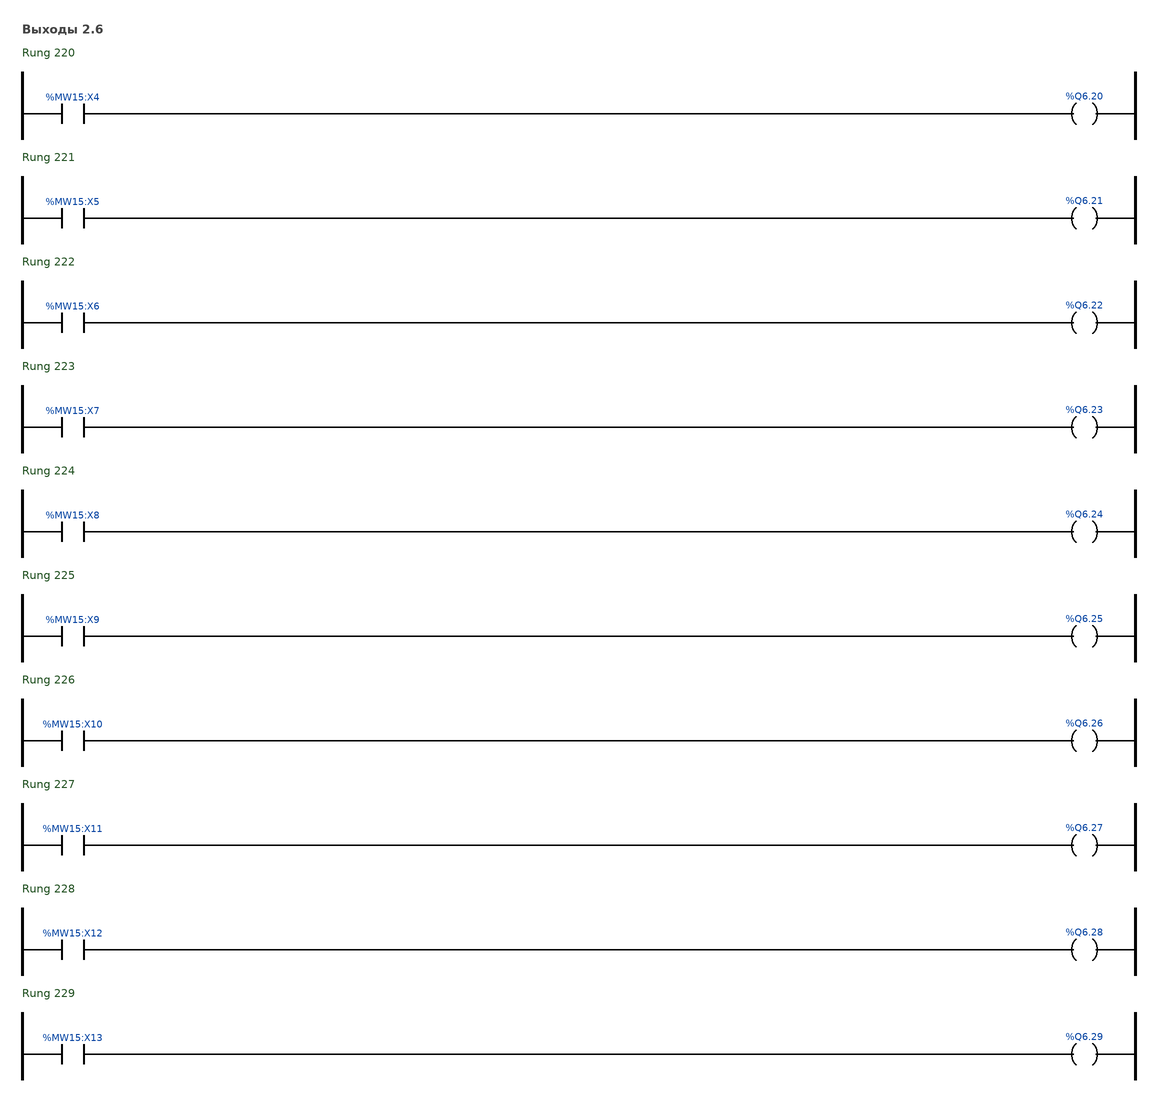

// Rung 220
  LD %MW15:X4
  ST %Q6.20
  // as ST:
  //   %Q6.20 := %MW15:X4;

// Rung 221
  LD %MW15:X5
  ST %Q6.21
  // as ST:
  //   %Q6.21 := %MW15:X5;

// Rung 222
  LD %MW15:X6
  ST %Q6.22
  // as ST:
  //   %Q6.22 := %MW15:X6;

// Rung 223
  LD %MW15:X7
  ST %Q6.23
  // as ST:
  //   %Q6.23 := %MW15:X7;

// Rung 224
  LD %MW15:X8
  ST %Q6.24
  // as ST:
  //   %Q6.24 := %MW15:X8;

// Rung 225
  LD %MW15:X9
  ST %Q6.25
  // as ST:
  //   %Q6.25 := %MW15:X9;

// Rung 226
  LD %MW15:X10
  ST %Q6.26
  // as ST:
  //   %Q6.26 := %MW15:X10;

// Rung 227
  LD %MW15:X11
  ST %Q6.27
  // as ST:
  //   %Q6.27 := %MW15:X11;

// Rung 228
  LD %MW15:X12
  ST %Q6.28
  // as ST:
  //   %Q6.28 := %MW15:X12;

// Rung 229
  LD %MW15:X13
  ST %Q6.29
  // as ST:
  //   %Q6.29 := %MW15:X13;

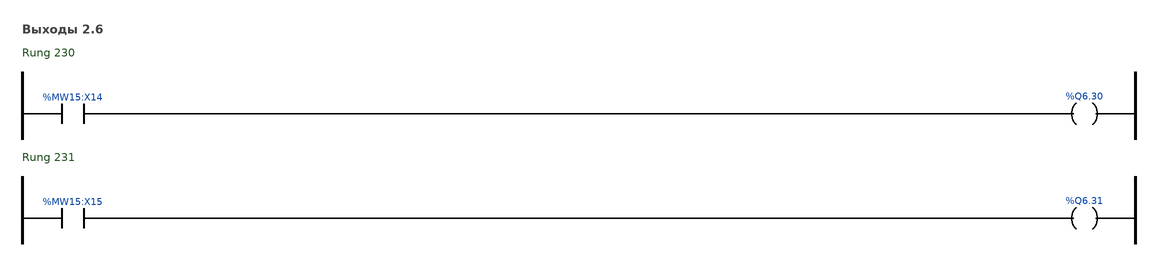

// Rung 230
  LD %MW15:X14
  ST %Q6.30
  // as ST:
  //   %Q6.30 := %MW15:X14;

// Rung 231
  LD %MW15:X15
  ST %Q6.31
  // as ST:
  //   %Q6.31 := %MW15:X15;

POU Выходы 2.7
  (* SectionNumber=9 *)

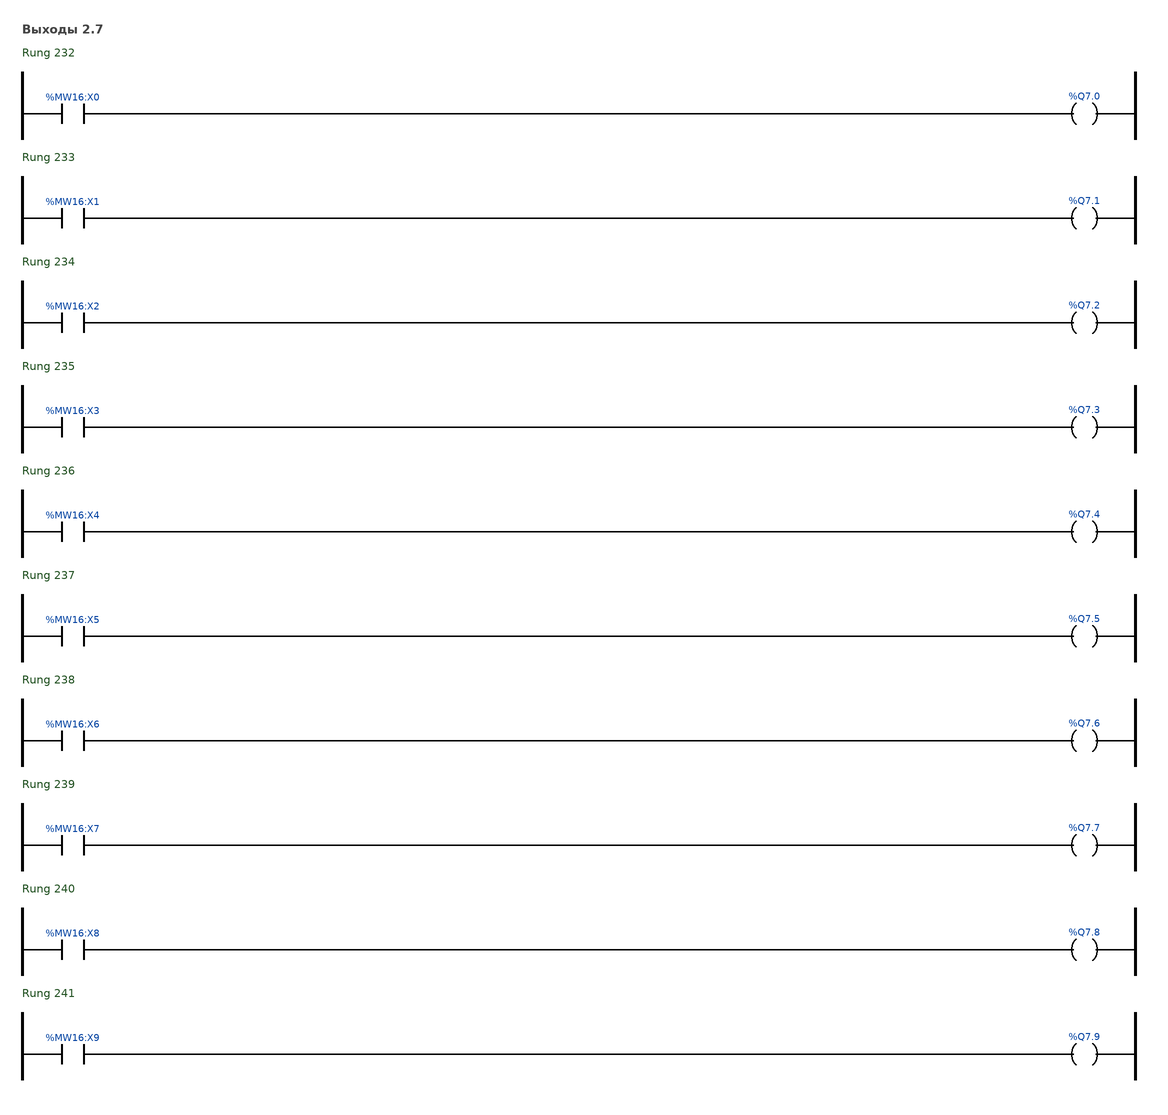

// Rung 232
  LD %MW16:X0
  ST %Q7.0
  // as ST:
  //   %Q7.0 := %MW16:X0;

// Rung 233
  LD %MW16:X1
  ST %Q7.1
  // as ST:
  //   %Q7.1 := %MW16:X1;

// Rung 234
  LD %MW16:X2
  ST %Q7.2
  // as ST:
  //   %Q7.2 := %MW16:X2;

// Rung 235
  LD %MW16:X3
  ST %Q7.3
  // as ST:
  //   %Q7.3 := %MW16:X3;

// Rung 236
  LD %MW16:X4
  ST %Q7.4
  // as ST:
  //   %Q7.4 := %MW16:X4;

// Rung 237
  LD %MW16:X5
  ST %Q7.5
  // as ST:
  //   %Q7.5 := %MW16:X5;

// Rung 238
  LD %MW16:X6
  ST %Q7.6
  // as ST:
  //   %Q7.6 := %MW16:X6;

// Rung 239
  LD %MW16:X7
  ST %Q7.7
  // as ST:
  //   %Q7.7 := %MW16:X7;

// Rung 240
  LD %MW16:X8
  ST %Q7.8
  // as ST:
  //   %Q7.8 := %MW16:X8;

// Rung 241
  LD %MW16:X9
  ST %Q7.9
  // as ST:
  //   %Q7.9 := %MW16:X9;

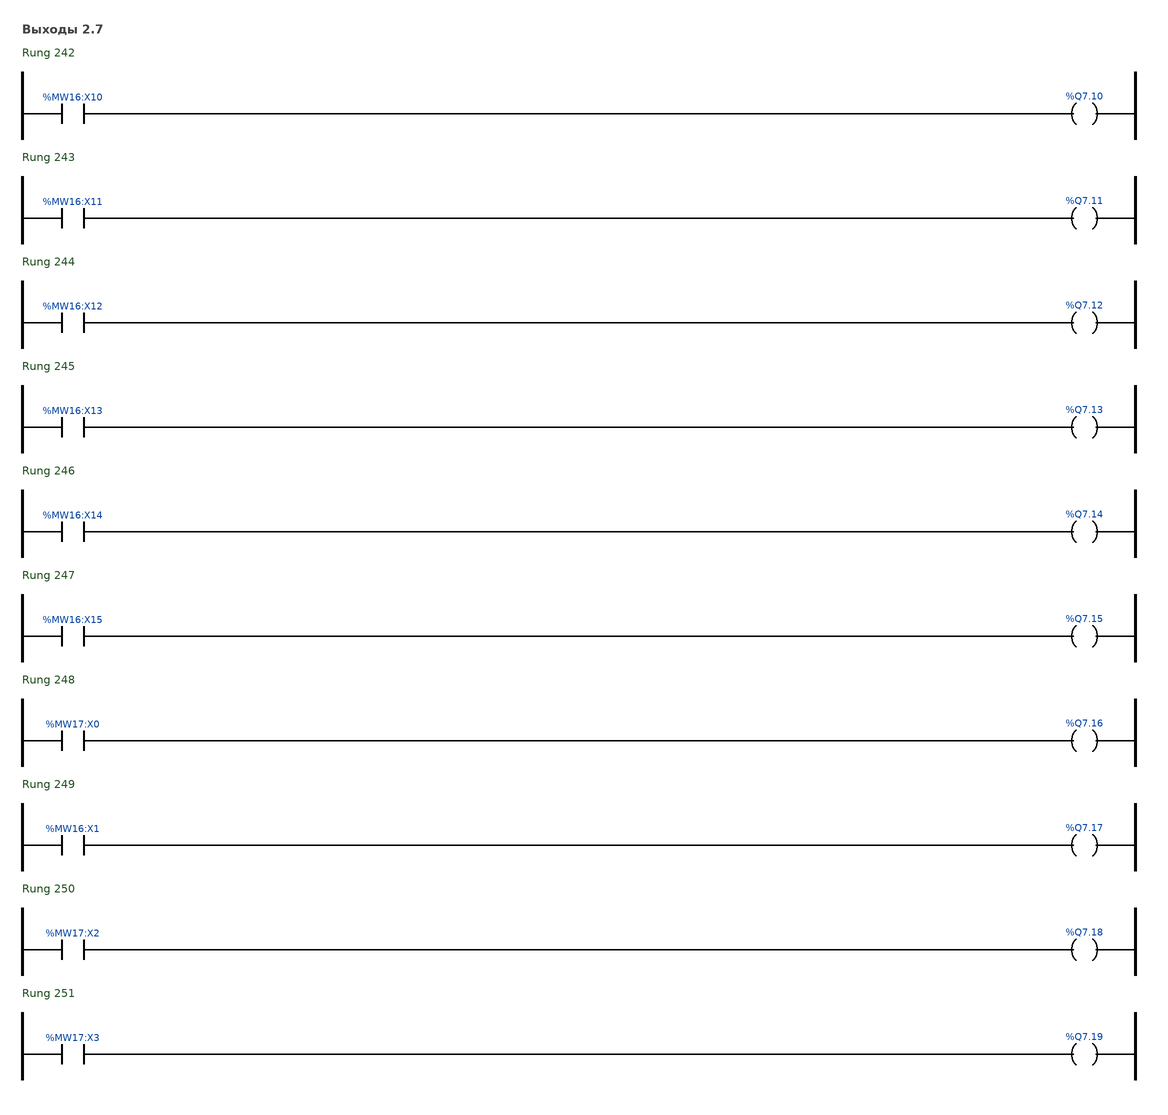

// Rung 242
  LD %MW16:X10
  ST %Q7.10
  // as ST:
  //   %Q7.10 := %MW16:X10;

// Rung 243
  LD %MW16:X11
  ST %Q7.11
  // as ST:
  //   %Q7.11 := %MW16:X11;

// Rung 244
  LD %MW16:X12
  ST %Q7.12
  // as ST:
  //   %Q7.12 := %MW16:X12;

// Rung 245
  LD %MW16:X13
  ST %Q7.13
  // as ST:
  //   %Q7.13 := %MW16:X13;

// Rung 246
  LD %MW16:X14
  ST %Q7.14
  // as ST:
  //   %Q7.14 := %MW16:X14;

// Rung 247
  LD %MW16:X15
  ST %Q7.15
  // as ST:
  //   %Q7.15 := %MW16:X15;

// Rung 248
  LD %MW17:X0
  ST %Q7.16
  // as ST:
  //   %Q7.16 := %MW17:X0;

// Rung 249
  LD %MW16:X1
  ST %Q7.17
  // as ST:
  //   %Q7.17 := %MW16:X1;

// Rung 250
  LD %MW17:X2
  ST %Q7.18
  // as ST:
  //   %Q7.18 := %MW17:X2;

// Rung 251
  LD %MW17:X3
  ST %Q7.19
  // as ST:
  //   %Q7.19 := %MW17:X3;

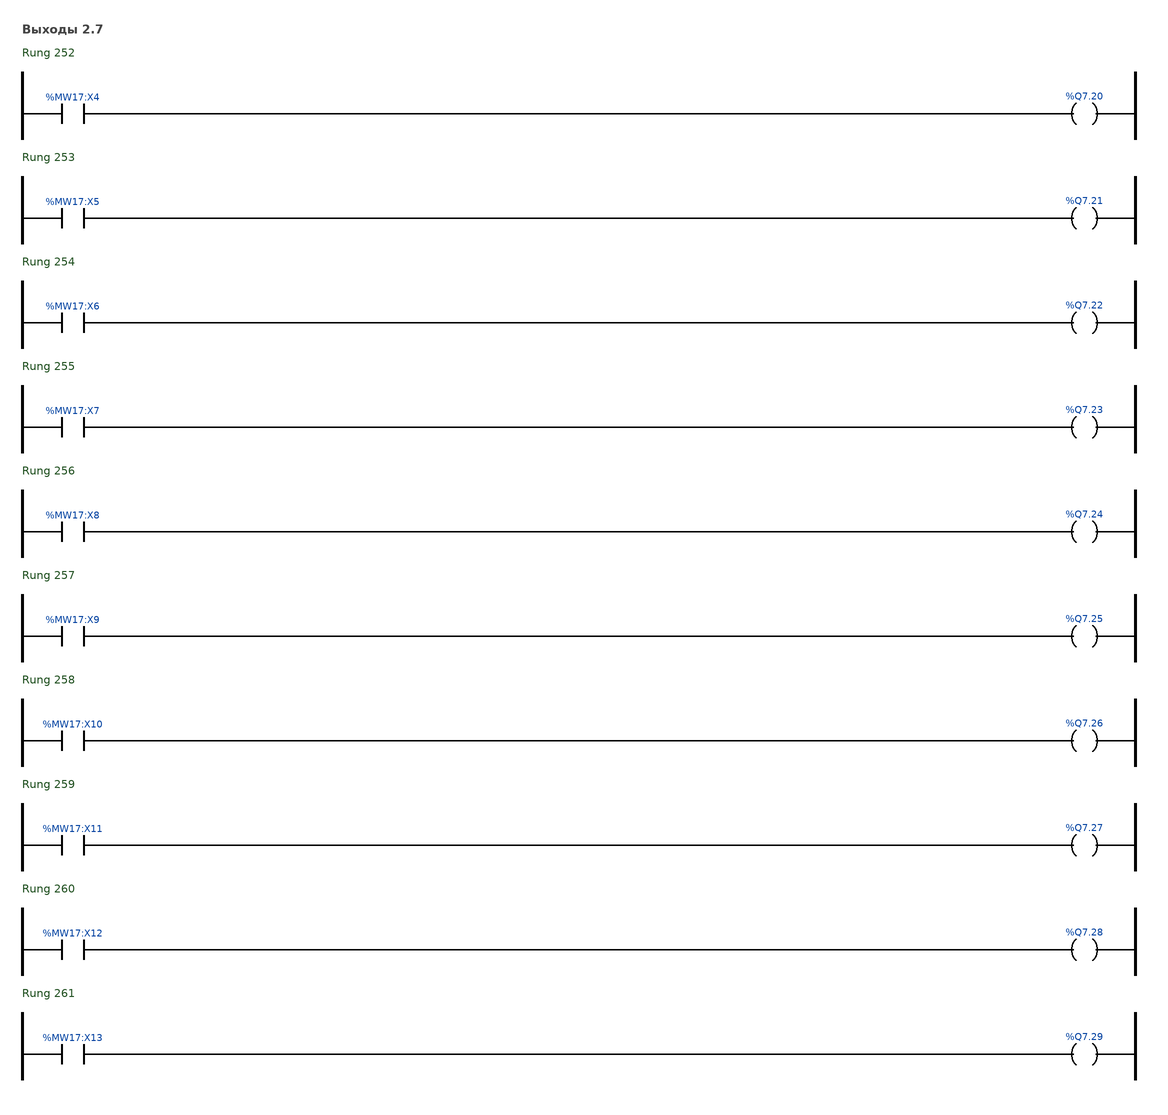

// Rung 252
  LD %MW17:X4
  ST %Q7.20
  // as ST:
  //   %Q7.20 := %MW17:X4;

// Rung 253
  LD %MW17:X5
  ST %Q7.21
  // as ST:
  //   %Q7.21 := %MW17:X5;

// Rung 254
  LD %MW17:X6
  ST %Q7.22
  // as ST:
  //   %Q7.22 := %MW17:X6;

// Rung 255
  LD %MW17:X7
  ST %Q7.23
  // as ST:
  //   %Q7.23 := %MW17:X7;

// Rung 256
  LD %MW17:X8
  ST %Q7.24
  // as ST:
  //   %Q7.24 := %MW17:X8;

// Rung 257
  LD %MW17:X9
  ST %Q7.25
  // as ST:
  //   %Q7.25 := %MW17:X9;

// Rung 258
  LD %MW17:X10
  ST %Q7.26
  // as ST:
  //   %Q7.26 := %MW17:X10;

// Rung 259
  LD %MW17:X11
  ST %Q7.27
  // as ST:
  //   %Q7.27 := %MW17:X11;

// Rung 260
  LD %MW17:X12
  ST %Q7.28
  // as ST:
  //   %Q7.28 := %MW17:X12;

// Rung 261
  LD %MW17:X13
  ST %Q7.29
  // as ST:
  //   %Q7.29 := %MW17:X13;

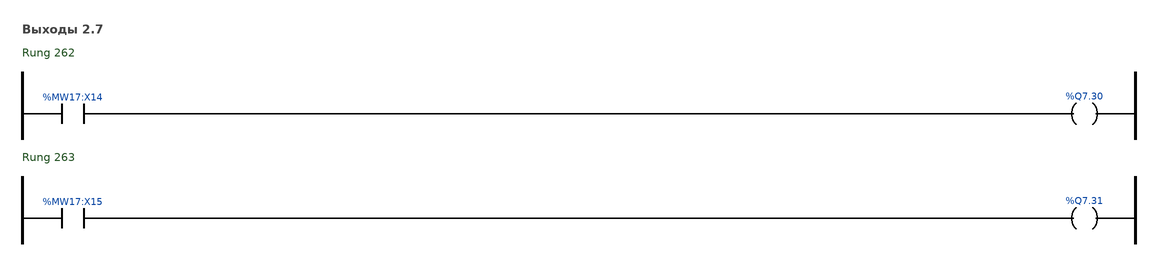

// Rung 262
  LD %MW17:X14
  ST %Q7.30
  // as ST:
  //   %Q7.30 := %MW17:X14;

// Rung 263
  LD %MW17:X15
  ST %Q7.31
  // as ST:
  //   %Q7.31 := %MW17:X15;

POU ДКС
  (* SectionNumber=10 *)

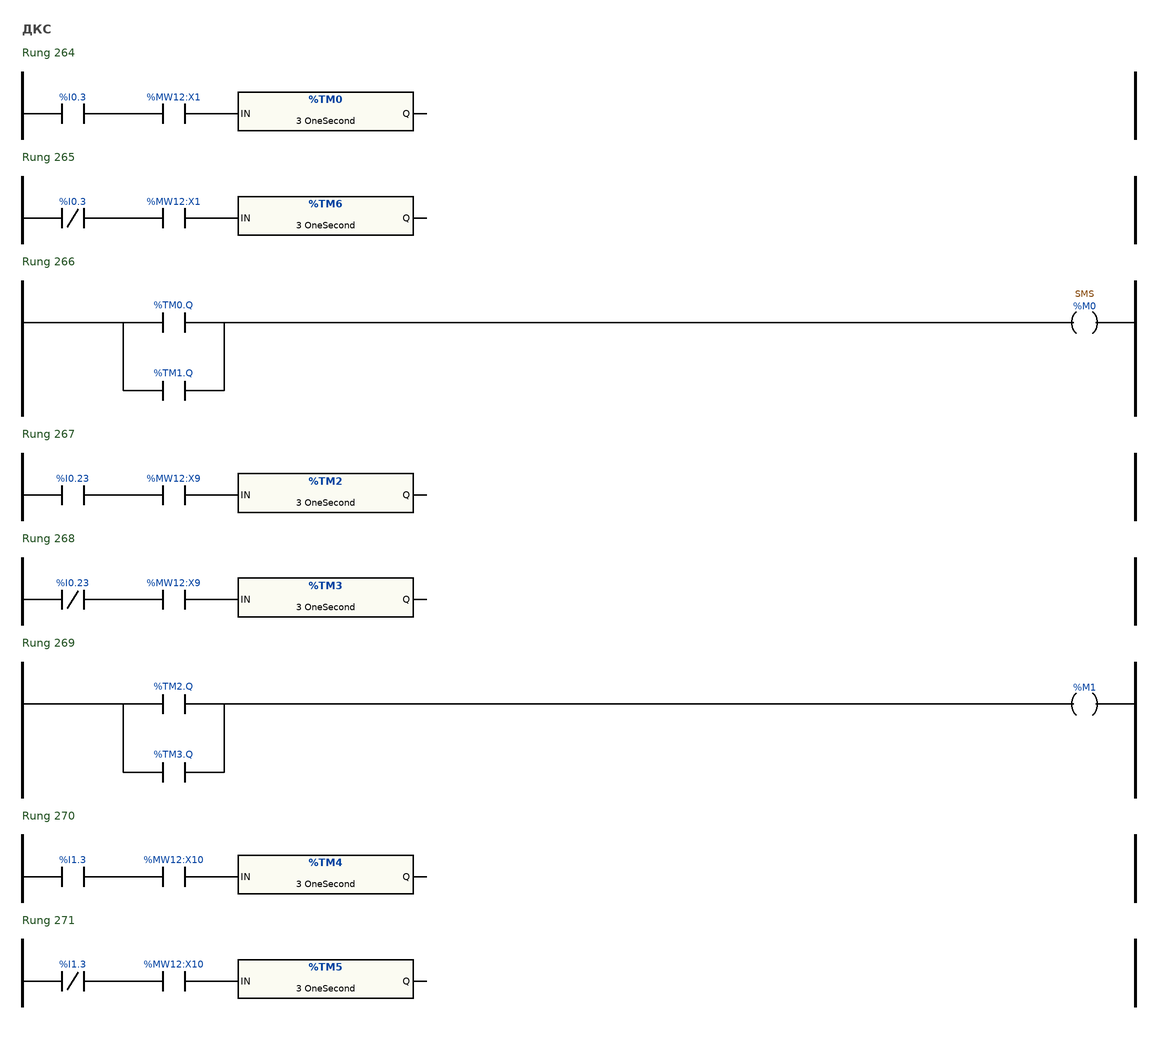

// Rung 264
  BLK %TM0
  LD %I0.3
  AND %MW12:X1
  IN
  END_BLK
  // as ST:
  //   %TM0(IN := %I0.3 AND %MW12:X1);

// Rung 265
  BLK %TM6
  LDN %I0.3
  AND %MW12:X1
  IN
  END_BLK
  // as ST:
  //   %TM6(IN := NOT %I0.3 AND %MW12:X1);

// Rung 266
  LD 1
  AND( %TM0.Q
  OR %TM1.Q
  )
  ST %M0                  (* SMS *)
  // as ST:
  //   SMS := %TM0.Q OR %TM1.Q;

// Rung 267
  BLK %TM2
  LD %I0.23
  AND %MW12:X9
  IN
  END_BLK
  // as ST:
  //   %TM2(IN := %I0.23 AND %MW12:X9);

// Rung 268
  BLK %TM3
  LDN %I0.23
  AND %MW12:X9
  IN
  END_BLK
  // as ST:
  //   %TM3(IN := NOT %I0.23 AND %MW12:X9);

// Rung 269
  LD 1
  AND( %TM2.Q
  OR %TM3.Q
  )
  ST %M1
  // as ST:
  //   %M1 := %TM2.Q OR %TM3.Q;

// Rung 270
  BLK %TM4
  LD %I1.3
  AND %MW12:X10
  IN
  END_BLK
  // as ST:
  //   %TM4(IN := %I1.3 AND %MW12:X10);

// Rung 271
  BLK %TM5
  LDN %I1.3
  AND %MW12:X10
  IN
  END_BLK
  // as ST:
  //   %TM5(IN := NOT %I1.3 AND %MW12:X10);

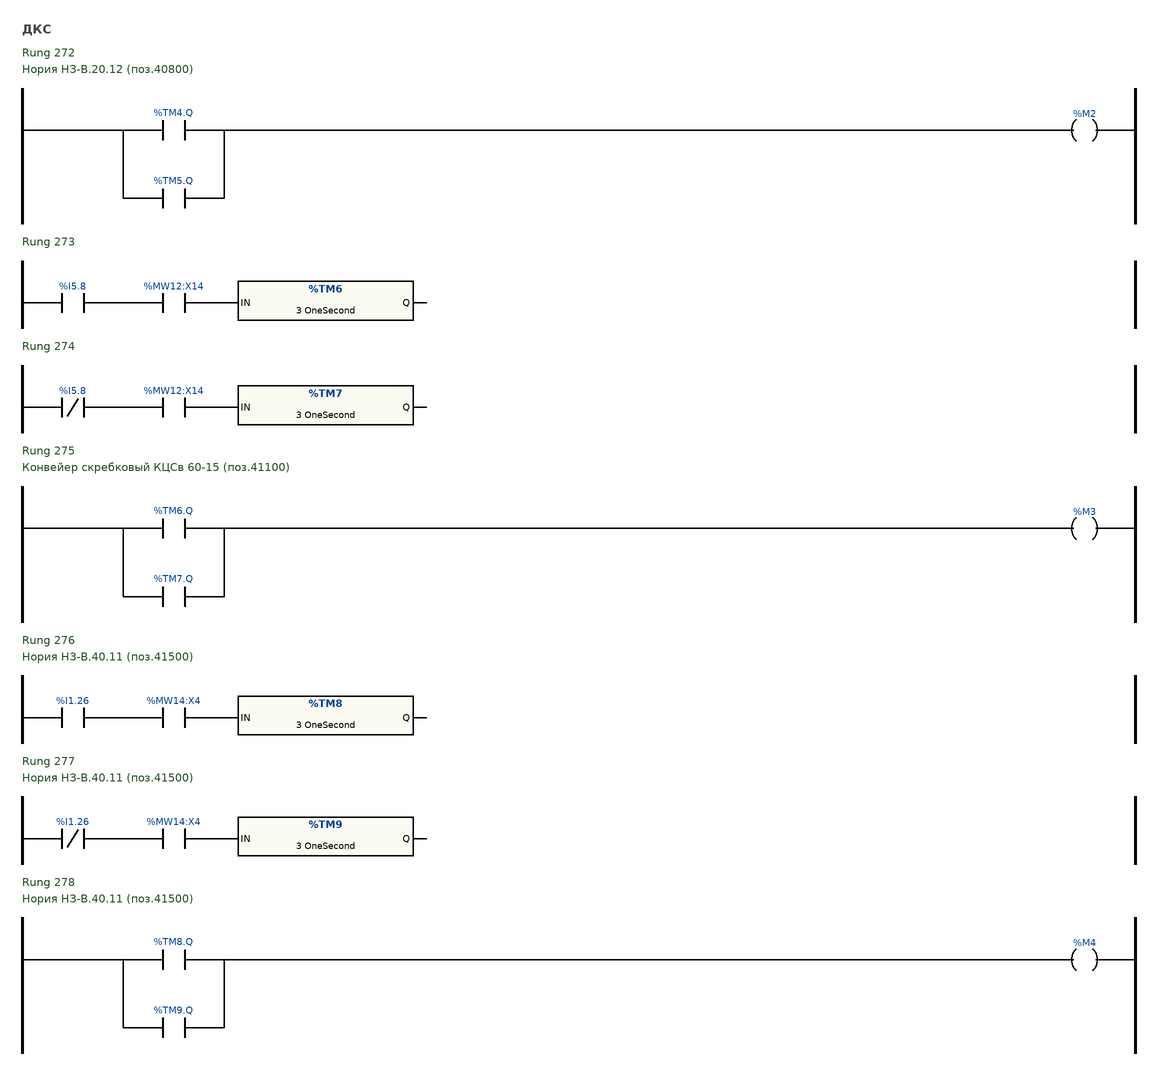

// Rung 272
// Нория НЗ-В.20.12 (поз.40800)
  LD 1
  AND( %TM4.Q
  OR %TM5.Q
  )
  ST %M2
  // as ST:
  //   %M2 := %TM4.Q OR %TM5.Q;

// Rung 273
  BLK %TM6
  LD %I5.8
  AND %MW12:X14
  IN
  END_BLK
  // as ST:
  //   %TM6(IN := %I5.8 AND %MW12:X14);

// Rung 274
  BLK %TM7
  LDN %I5.8
  AND %MW12:X14
  IN
  END_BLK
  // as ST:
  //   %TM7(IN := NOT %I5.8 AND %MW12:X14);

// Rung 275
// Конвейер скребковый КЦСв 60-15 (поз.41100)
  LD 1
  AND( %TM6.Q
  OR %TM7.Q
  )
  ST %M3
  // as ST:
  //   %M3 := %TM6.Q OR %TM7.Q;

// Rung 276
// Нория НЗ-В.40.11 (поз.41500)
  BLK %TM8
  LD %I1.26
  AND %MW14:X4
  IN
  END_BLK
  // as ST:
  //   %TM8(IN := %I1.26 AND %MW14:X4);

// Rung 277
// Нория НЗ-В.40.11 (поз.41500)
  BLK %TM9
  LDN %I1.26
  AND %MW14:X4
  IN
  END_BLK
  // as ST:
  //   %TM9(IN := NOT %I1.26 AND %MW14:X4);

// Rung 278
// Нория НЗ-В.40.11 (поз.41500)
  LD 1
  AND( %TM8.Q
  OR %TM9.Q
  )
  ST %M4
  // as ST:
  //   %M4 := %TM8.Q OR %TM9.Q;

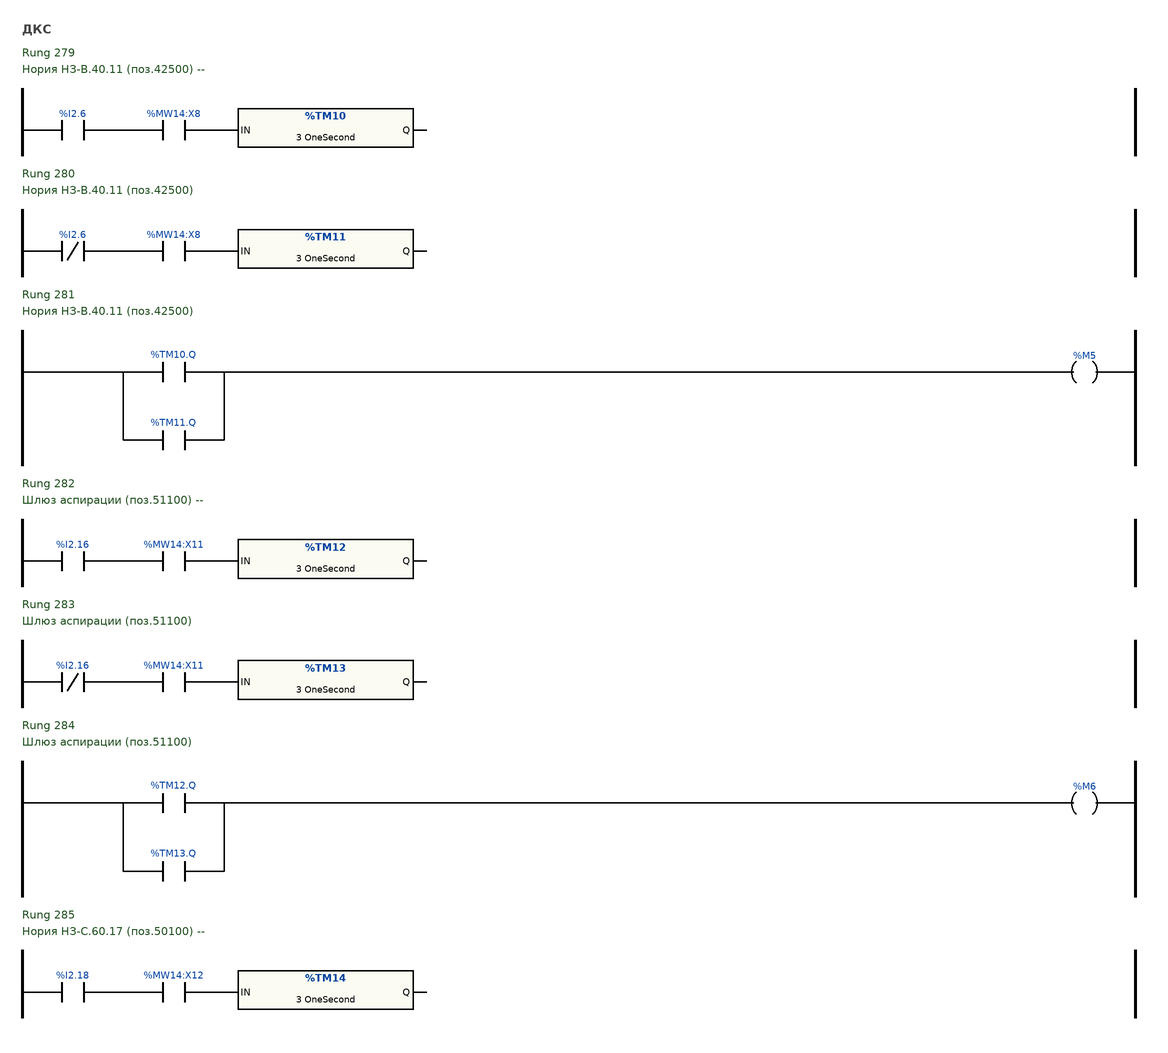

// Rung 279
// Нория НЗ-В.40.11 (поз.42500) --
  BLK %TM10
  LD %I2.6
  AND %MW14:X8
  IN
  END_BLK
  // as ST:
  //   %TM10(IN := %I2.6 AND %MW14:X8);

// Rung 280
// Нория НЗ-В.40.11 (поз.42500)
  BLK %TM11
  LDN %I2.6
  AND %MW14:X8
  IN
  END_BLK
  // as ST:
  //   %TM11(IN := NOT %I2.6 AND %MW14:X8);

// Rung 281
// Нория НЗ-В.40.11 (поз.42500)
  LD 1
  AND( %TM10.Q
  OR %TM11.Q
  )
  ST %M5
  // as ST:
  //   %M5 := %TM10.Q OR %TM11.Q;

// Rung 282
// Шлюз аспирации (поз.51100) --
  BLK %TM12
  LD %I2.16
  AND %MW14:X11
  IN
  END_BLK
  // as ST:
  //   %TM12(IN := %I2.16 AND %MW14:X11);

// Rung 283
// Шлюз аспирации (поз.51100)
  BLK %TM13
  LDN %I2.16
  AND %MW14:X11
  IN
  END_BLK
  // as ST:
  //   %TM13(IN := NOT %I2.16 AND %MW14:X11);

// Rung 284
// Шлюз аспирации (поз.51100)
  LD 1
  AND( %TM12.Q
  OR %TM13.Q
  )
  ST %M6
  // as ST:
  //   %M6 := %TM12.Q OR %TM13.Q;

// Rung 285
// Нория НЗ-С.60.17 (поз.50100) --
  BLK %TM14
  LD %I2.18
  AND %MW14:X12
  IN
  END_BLK
  // as ST:
  //   %TM14(IN := %I2.18 AND %MW14:X12);

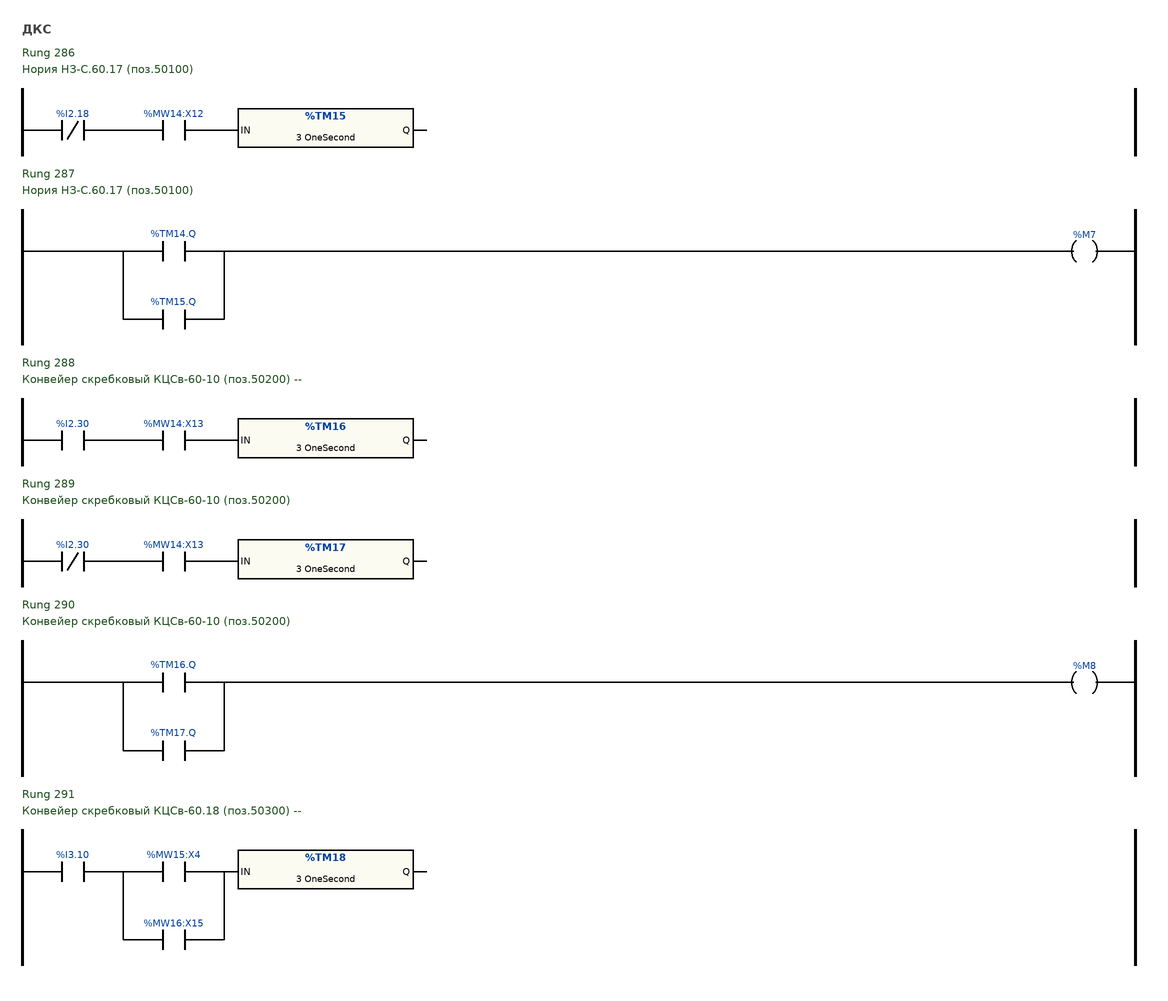

// Rung 286
// Нория НЗ-С.60.17 (поз.50100)
  BLK %TM15
  LDN %I2.18
  AND %MW14:X12
  IN
  END_BLK
  // as ST:
  //   %TM15(IN := NOT %I2.18 AND %MW14:X12);

// Rung 287
// Нория НЗ-С.60.17 (поз.50100)
  LD 1
  AND( %TM14.Q
  OR %TM15.Q
  )
  ST %M7
  // as ST:
  //   %M7 := %TM14.Q OR %TM15.Q;

// Rung 288
// Конвейер скребковый КЦСв-60-10 (поз.50200) --
  BLK %TM16
  LD %I2.30
  AND %MW14:X13
  IN
  END_BLK
  // as ST:
  //   %TM16(IN := %I2.30 AND %MW14:X13);

// Rung 289
// Конвейер скребковый КЦСв-60-10 (поз.50200)
  BLK %TM17
  LDN %I2.30
  AND %MW14:X13
  IN
  END_BLK
  // as ST:
  //   %TM17(IN := NOT %I2.30 AND %MW14:X13);

// Rung 290
// Конвейер скребковый КЦСв-60-10 (поз.50200)
  LD 1
  AND( %TM16.Q
  OR %TM17.Q
  )
  ST %M8
  // as ST:
  //   %M8 := %TM16.Q OR %TM17.Q;

// Rung 291
// Конвейер скребковый КЦСв-60.18 (поз.50300) --
  BLK %TM18
  LD %I3.10
  AND( %MW15:X4
  OR %MW16:X15
  )
  IN
  END_BLK
  // as ST:
  //   %TM18(IN := %I3.10 AND (%MW15:X4 OR %MW16:X15));

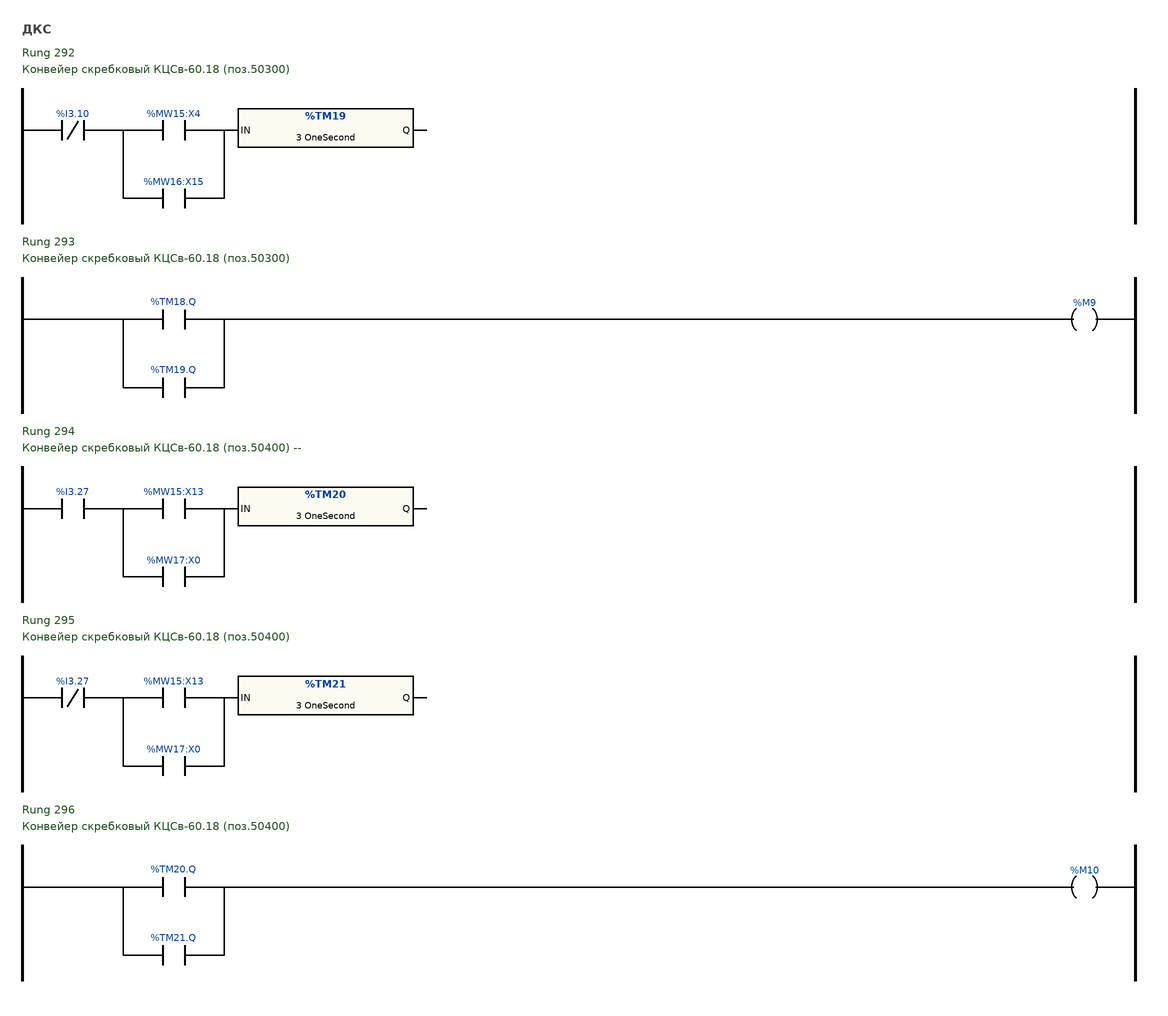

// Rung 292
// Конвейер скребковый КЦСв-60.18 (поз.50300)
  BLK %TM19
  LDN %I3.10
  AND( %MW15:X4
  OR %MW16:X15
  )
  IN
  END_BLK
  // as ST:
  //   %TM19(IN := NOT %I3.10 AND (%MW15:X4 OR %MW16:X15));

// Rung 293
// Конвейер скребковый КЦСв-60.18 (поз.50300)
  LD 1
  AND( %TM18.Q
  OR %TM19.Q
  )
  ST %M9
  // as ST:
  //   %M9 := %TM18.Q OR %TM19.Q;

// Rung 294
// Конвейер скребковый КЦСв-60.18 (поз.50400) --
  BLK %TM20
  LD %I3.27
  AND( %MW15:X13
  OR %MW17:X0
  )
  IN
  END_BLK
  // as ST:
  //   %TM20(IN := %I3.27 AND (%MW15:X13 OR %MW17:X0));

// Rung 295
// Конвейер скребковый КЦСв-60.18 (поз.50400)
  BLK %TM21
  LDN %I3.27
  AND( %MW15:X13
  OR %MW17:X0
  )
  IN
  END_BLK
  // as ST:
  //   %TM21(IN := NOT %I3.27 AND (%MW15:X13 OR %MW17:X0));

// Rung 296
// Конвейер скребковый КЦСв-60.18 (поз.50400)
  LD 1
  AND( %TM20.Q
  OR %TM21.Q
  )
  ST %M10
  // as ST:
  //   %M10 := %TM20.Q OR %TM21.Q;

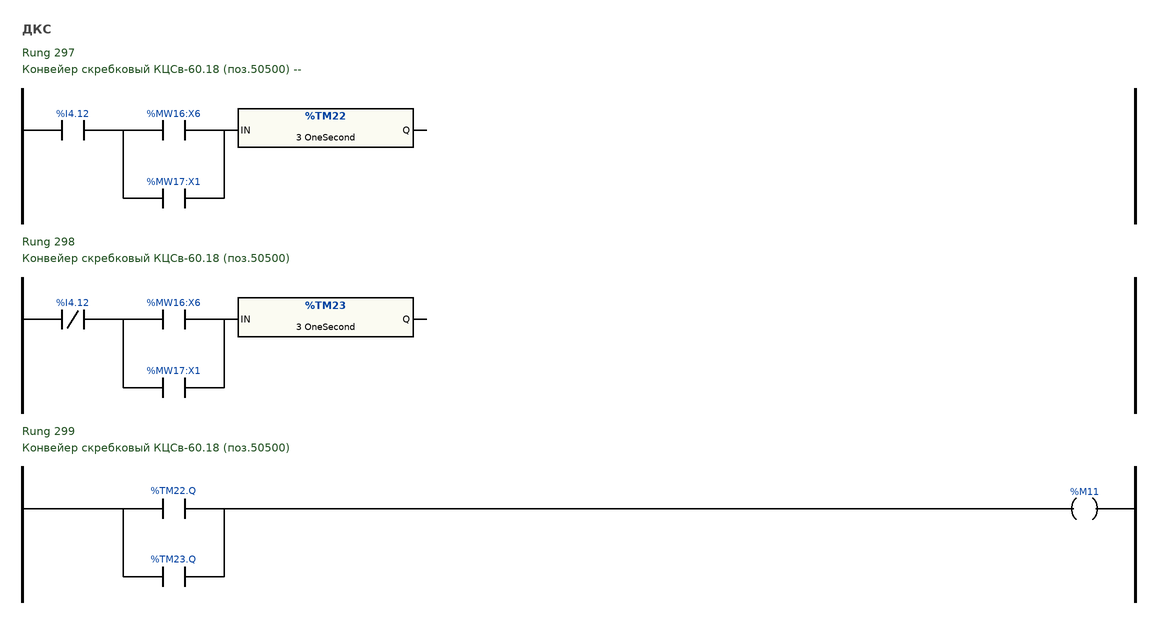

// Rung 297
// Конвейер скребковый КЦСв-60.18 (поз.50500) --
  BLK %TM22
  LD %I4.12
  AND( %MW16:X6
  OR %MW17:X1
  )
  IN
  END_BLK
  // as ST:
  //   %TM22(IN := %I4.12 AND (%MW16:X6 OR %MW17:X1));

// Rung 298
// Конвейер скребковый КЦСв-60.18 (поз.50500)
  BLK %TM23
  LDN %I4.12
  AND( %MW16:X6
  OR %MW17:X1
  )
  IN
  END_BLK
  // as ST:
  //   %TM23(IN := NOT %I4.12 AND (%MW16:X6 OR %MW17:X1));

// Rung 299
// Конвейер скребковый КЦСв-60.18 (поз.50500)
  LD 1
  AND( %TM22.Q
  OR %TM23.Q
  )
  ST %M11
  // as ST:
  //   %M11 := %TM22.Q OR %TM23.Q;
